PROGRAM MAIN
VAR
END_VAR

END_PROGRAM

(* stored: Version 1.1.0.1, ProductVersion 3.1.0.36
   POU MAIN: Id {e418c60e-009c-4d8f-b608-e5fd93d22680}, SpecialFunc None *)
